VAR_GLOBAL
//	stWrite				AT%MB0		: ST_Communication;			//Wysyłane zmienne do BottleUnboxer
//	stRead				AT%I*		: ST_Communication;			//Odczytane zmienne z BottleUnboxer

	// Sygnały pomocnicze
	bEnable									: BOOL;
	bCycleStart								: BOOL;
	bCycleStop								: BOOL;
	bCycleReset								: BOOL;
	bManualMode								: BOOL;
	bHoming									: BOOL;	
	bHomingDone								: BOOL;
	bConfectionEnding						: BOOL;	
	bHomingDialog							: BOOL;
	bHomingCanceled							: BOOL;
	bChooseRecipe							: BOOL;
	bSafetyState							: BOOL;
	bReset									: BOOL;					// reset bledow z XTS          
	bRunLock								: BOOL;					//Blokada pracy   
	bSafetyReset							: BOOL;   
	bRecipeLoading							: BOOL;					//Wystawiane jak receptura jest ładowana                                           	
	bEmptingMode							: BOOL;
	bDoorClose								: BOOL;
END_VAR

(* stored: Version 1.1.0.1, FileIdentifier 712735cafe4a70a78aa0caa1292f8cd8c0fbbccd, FileSignature 720fa911cfddbd551f0cdcbc264012281fd7ce2ee9cb4f90f74bb9f4d80f589051a9584e2ca39c9c124c6e1fbd774add9a271d49a45c9d014348227d176de4dba975586344d426d7997c5bbf281c6e0b8d945e877c99e36c66213e2053c5130ef5c5728d4a8d634a884fe1765ac06eb4ef4948458a415070a26ac365f579b29486c75a75ced7812e580291e4231b9a1ea18ed5cfa0dce4c57bb89ee99fb7452390053d1832a61dedc316441afdb964e5b7b39050a9a10d939e4b5583e670ea4985f408ded3bb2e372b8ab684bf6ff9b4d6f27804e46b842b0f48d7c5884ba7c880eedaa98bdc757695cee34d7dad9aaec03578644b2b17e2118c388578cfabd7
   GVL GVL_Communication: Id {75259b54-1b00-422f-b035-f9ad055d0c01} *)
